FUNCTION_BLOCK t (* Basic FB with empty ECC *)
  (* Standard: 61499-2; Description: Part of ellipse fitting method block function, to find t. *)
  (* Version 1.0, 2020-08-17, Candra Wardaya, UGM *)
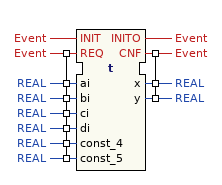
  EVENT_INPUT
    INIT;
    REQ WITH ai, bi, ci, di, const_4, const_5;
  END_EVENT
  EVENT_OUTPUT
    INITO;
    CNF WITH x, y;
  END_EVENT
  VAR_INPUT
    ai : REAL;
    bi : REAL;
    ci : REAL;
    di : REAL;
    const_4 : REAL;
    const_5 : REAL;
  END_VAR
  VAR_OUTPUT
    x : REAL;
    y : REAL;
  END_VAR
  VAR
    xi : REAL; (* Internal Variable *)
    yi : REAL; (* Internal Variable *)
  END_VAR
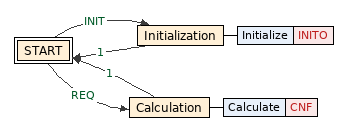
  EC_STATES
    START; (* Initial State *)
    Initialization : Initialize -> INITO;
    Calculation : Calculate -> CNF;
  END_STATES
  EC_TRANSITIONS
    START TO Initialization := INIT;
    Initialization TO START := 1;
    START TO Calculation := REQ;
    Calculation TO START := 1;
  END_TRANSITIONS
  ALGORITHM Initialize IN ST: (* New Algorithm *)

  END_ALGORITHM
  ALGORITHM Calculate IN ST: (* New Algorithm *)
xi := ai*const_4 + bi*const_5;
yi := ci*const_4 + di*const_5;

x := -0.5*xi;
y := -0.5*yi;
  END_ALGORITHM
END_FUNCTION_BLOCK
